(* Logix 5000 project; controller Google vendor 1 type 14 code 151 rev 31.11; software revision 31.00; part 6 of 6 *)
(* tags used below, declared in another part *)
   Alarm : BOOL[64];
   Alarm_Active : BOOL;
   Alarm_Delay : TIMER[32];
   Alarm_Horn : BOOL;
   Alarm_Pulser : Pulser;
   Alarm_Silence : BOOL;
   E_Stop_Pressed : BOOL;
   HMI_Alarm_Silence : BOOL;
   HMI_AutoMode : BOOL;
   HMI_Conv_FWD_Speed : DINT;
   HMI_Conv_REV_Speed : DINT;
   HMI_Conv_Start_Delay : DINT;
   HMI_JogMode : BOOL;
   HMI_ManualMode : BOOL;
   HMI_Output1 : BOOL[32];
   HMI_OutputTest : BOOL[32];
   HMI_PB_Reset : BOOL;
   HMI_System_Full : BOOL;
   Infeed_Conv_Motors : Conveyor_Motor_Control;
   Infeed_ModuleFaultCode : DINT;
   Infeed_Zone1_FWD : BOOL;
   Infeed_Zone1_REV : BOOL;
   Infeed_Zone2_FWD : BOOL;
   Infeed_Zone2_REV : BOOL;
   Infeed_Zone3_FWD : BOOL;
   Infeed_Zone3_REV : BOOL;
   Infeed_Zone4_FWD : BOOL;
   Infeed_Zone4_REV : BOOL;
   L1_Conv_Motors : Conveyor_Motor_Control;
   L1_ModuleFaultCode : DINT;
   L1_Zone1_FWD : BOOL;
   L1_Zone1_REV : BOOL;
   L1_Zone2_FWD : BOOL;
   L1_Zone2_REV : BOOL;
   L1_Zone3_FWD : BOOL;
   L1_Zone3_REV : BOOL;
   L1_Zone4_FWD : BOOL;
   L1_Zone4_REV : BOOL;
   L2_Conv_Motors : Conveyor_Motor_Control;
   L2_ModuleFaultCode : DINT;
   L2_Zone1_FWD : BOOL;
   L2_Zone1_REV : BOOL;
   L2_Zone2_FWD : BOOL;
   L2_Zone2_REV : BOOL;
   L2_Zone3_FWD : BOOL;
   L2_Zone3_REV : BOOL;
   L2_Zone4_FWD : BOOL;
   L2_Zone4_REV : BOOL;
   L3_Conv_Motors : Conveyor_Motor_Control;
   L3_ModuleFaultCode : DINT;
   L3_Zone1_FWD : BOOL;
   L3_Zone1_REV : BOOL;
   L3_Zone2_FWD : BOOL;
   L3_Zone2_REV : BOOL;
   L3_Zone3_FWD : BOOL;
   L3_Zone3_REV : BOOL;
   L3_Zone4_FWD : BOOL;
   L3_Zone4_REV : BOOL;
   L4_Conv_Motors : Conveyor_Motor_Control;
   L4_ModuleFaultCode : DINT;
   L4_Zone1_FWD : BOOL;
   L4_Zone1_REV : BOOL;
   L4_Zone2_FWD : BOOL;
   L4_Zone2_REV : BOOL;
   L4_Zone3_FWD : BOOL;
   L4_Zone3_REV : BOOL;
   L4_Zone4_FWD : BOOL;
   L4_Zone4_REV : BOOL;
   L5_Conv_Motors : Conveyor_Motor_Control;
   L5_ModuleFaultCode : DINT;
   L5_Zone1_FWD : BOOL;
   L5_Zone1_REV : BOOL;
   L5_Zone2_FWD : BOOL;
   L5_Zone2_REV : BOOL;
   L5_Zone3_FWD : BOOL;
   L5_Zone3_REV : BOOL;
   L5_Zone4_FWD : BOOL;
   L5_Zone4_REV : BOOL;
   Level_2_Full : BOOL;
   Level_3_Full : BOOL;
   Level_4_Full : BOOL;
   Level_5_Full : BOOL;
   Lift_Alarm : BOOL;
   Lift_Conv_Motor : Lift_Conv_Motor_Control;
   Lift_ModuleFaultCode : DINT;
   LiftZone_FWD : BOOL;
   LiftZone_REV : BOOL;
   Manual_Mode_Active : BOOL;
   MCR_DelayActive : BOOL;
   MCR_Enable : BOOL;
   MCR_EnableDelay : TIMER;
   MCR_Status : BOOL;
   ONS : DINT[6];
   Outputs_1 : Output_16_Bit;
   PS10017_DC_OK : BOOL;
   Ready_Pulser : Pulser;
   Safety_OK : BOOL;
   Safety_OK_Delay : TIMER;
   Safety_Relay_Status : BOOL;
   Spare_Output : BOOL;
   Stacklight_Amber : BOOL;
   Stacklight_Audible : BOOL;
   Stacklight_Green : BOOL;
   Stacklight_Red : BOOL;
   Starting_Horn : BOOL;
   Starting_Pulser : Pulser;
   Stopping_Pulser : Pulser;
   System : State;
   System_State : DINT;
(* MainProgram, continued *)

ROUTINE R14_Stacklight   (* ladder *)
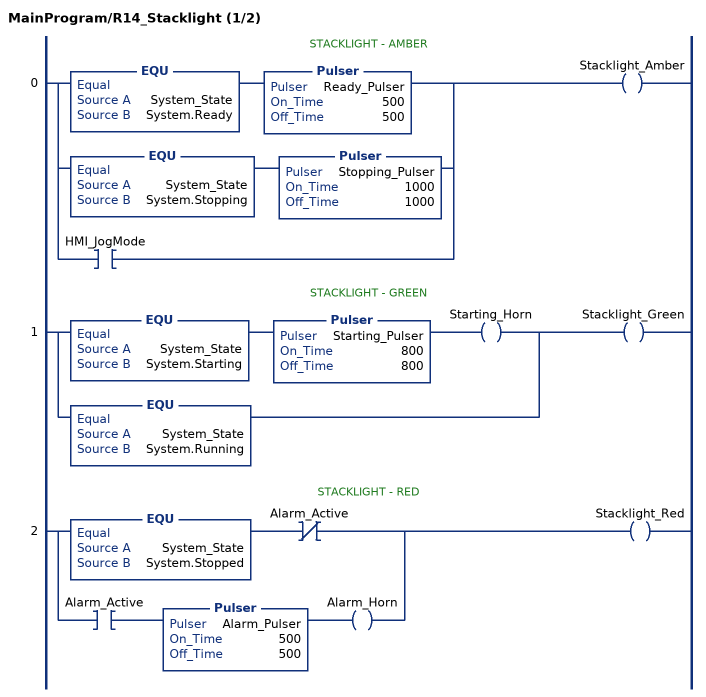
   // STACKLIGHT - AMBER
   0: [EQU(System_State,System.Ready) Pulser(Ready_Pulser,500,500) ,EQU(System_State,System.Stopping) Pulser(Stopping_Pulser,1000,1000) ,XIC(HMI_JogMode) ]OTE(Stacklight_Amber);
   // STACKLIGHT - GREEN
   1: [EQU(System_State,System.Starting) Pulser(Starting_Pulser,800,800) OTE(Starting_Horn) ,EQU(System_State,System.Running) ]OTE(Stacklight_Green);
   // STACKLIGHT - RED
   2: [EQU(System_State,System.Stopped) XIO(Alarm_Active) ,XIC(Alarm_Active) Pulser(Alarm_Pulser,500,500) OTE(Alarm_Horn) ]OTE(Stacklight_Red);
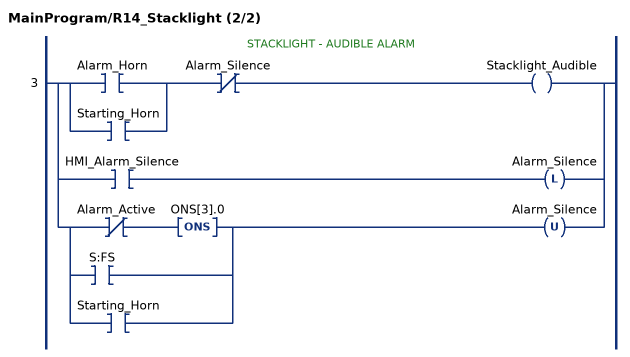
   // STACKLIGHT - AUDIBLE ALARM
   3: [[XIC(Alarm_Horn) ,XIC(Starting_Horn) ] XIO(Alarm_Silence) OTE(Stacklight_Audible) ,XIC(HMI_Alarm_Silence) OTL(Alarm_Silence) ,[XIO(Alarm_Active) ONS(ONS[3].0) ,XIC(S:FS) ,XIC(Starting_Horn) ] OTU(Alarm_Silence) ];
END_ROUTINE

ROUTINE R15_Alarms   (* ladder *)
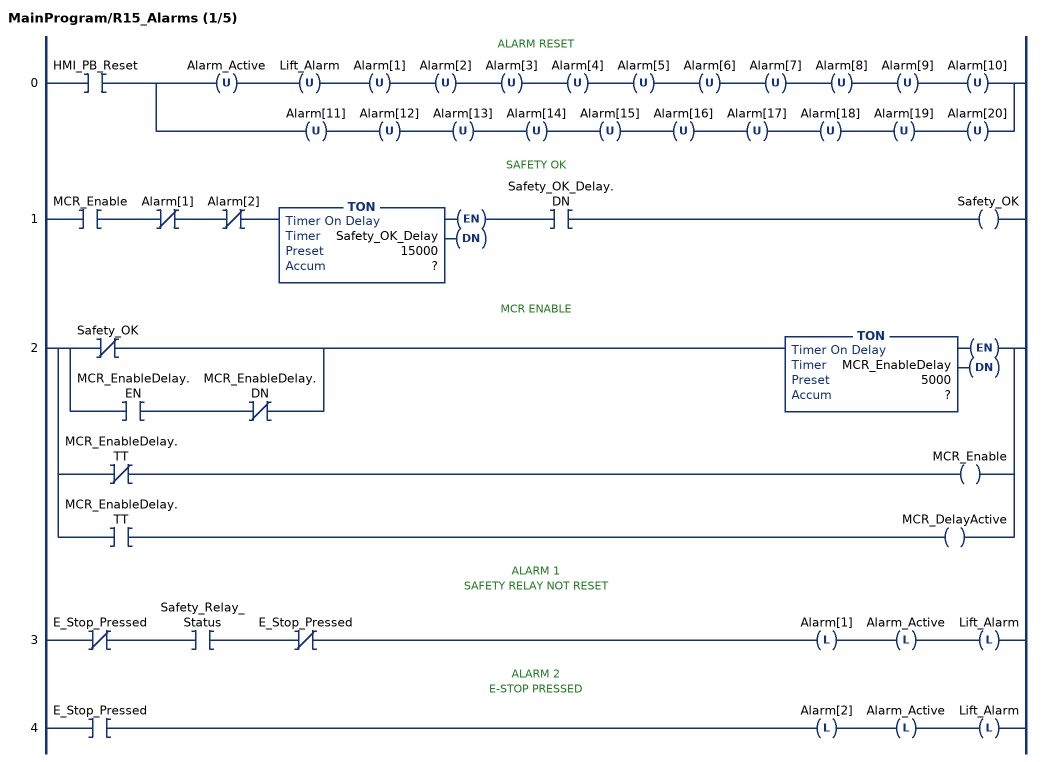
   // ALARM RESET
   0: XIC(HMI_PB_Reset)[OTU(Alarm_Active) OTU(Lift_Alarm) OTU(Alarm[1]) OTU(Alarm[2]) OTU(Alarm[3]) OTU(Alarm[4]) OTU(Alarm[5]) OTU(Alarm[6]) OTU(Alarm[7]) OTU(Alarm[8]) OTU(Alarm[9]) OTU(Alarm[10]) ,OTU(Alarm[11]) OTU(Alarm[12]) OTU(Alarm[13]) OTU(Alarm[14]) OTU(Alarm[15]) OTU(Alarm[16]) OTU(Alarm[17]) OTU(Alarm[18]) OTU(Alarm[19]) OTU(Alarm[20]) ];
   // SAFETY OK
   1: XIC(MCR_Enable)XIO(Alarm[1])XIO(Alarm[2])TON(Safety_OK_Delay,?,?)XIC(Safety_OK_Delay.DN)OTE(Safety_OK);
   // MCR ENABLE
   2: [[XIO(Safety_OK) ,XIC(MCR_EnableDelay.EN) XIO(MCR_EnableDelay.DN) ] TON(MCR_EnableDelay,?,?) ,XIO(MCR_EnableDelay.TT) OTE(MCR_Enable) ,XIC(MCR_EnableDelay.TT) OTE(MCR_DelayActive) ];
   // ALARM 1
   // SAFETY RELAY NOT RESET
   3: XIO(E_Stop_Pressed)XIC(Safety_Relay_Status)XIO(E_Stop_Pressed)OTL(Alarm[1])OTL(Alarm_Active)OTL(Lift_Alarm);
   // ALARM 2
   // E-STOP PRESSED
   4: XIC(E_Stop_Pressed)OTL(Alarm[2])OTL(Alarm_Active)OTL(Lift_Alarm);
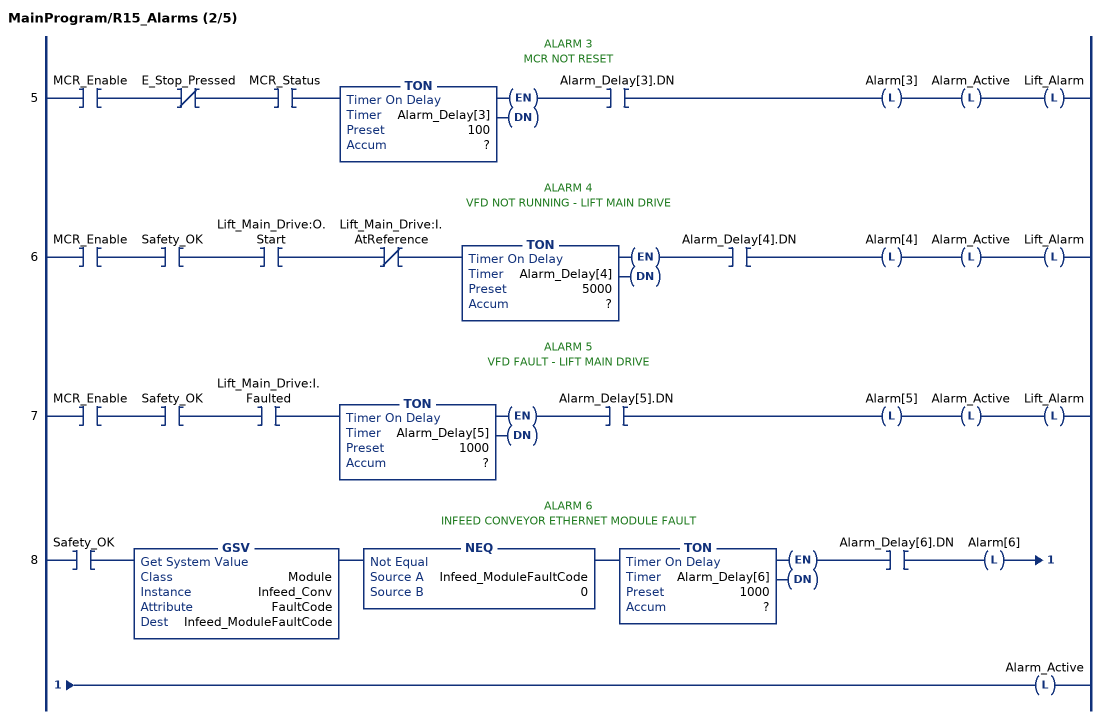
   // ALARM 3
   // MCR NOT RESET
   5: XIC(MCR_Enable)XIO(E_Stop_Pressed)XIC(MCR_Status)TON(Alarm_Delay[3],?,?)XIC(Alarm_Delay[3].DN)OTL(Alarm[3])OTL(Alarm_Active)OTL(Lift_Alarm);
   // ALARM 4
   // VFD NOT RUNNING - LIFT MAIN DRIVE
   6: XIC(MCR_Enable)XIC(Safety_OK)XIC(Lift_Main_Drive:O.Start)XIO(Lift_Main_Drive:I.AtReference)TON(Alarm_Delay[4],?,?)XIC(Alarm_Delay[4].DN)OTL(Alarm[4])OTL(Alarm_Active)OTL(Lift_Alarm);
   // ALARM 5
   // VFD FAULT - LIFT MAIN DRIVE
   7: XIC(MCR_Enable)XIC(Safety_OK)XIC(Lift_Main_Drive:I.Faulted)TON(Alarm_Delay[5],?,?)XIC(Alarm_Delay[5].DN)OTL(Alarm[5])OTL(Alarm_Active)OTL(Lift_Alarm);
   // ALARM 6
   // INFEED CONVEYOR ETHERNET MODULE FAULT
   8: XIC(Safety_OK)GSV(Module,Infeed_Conv,FaultCode,Infeed_ModuleFaultCode)NEQ(Infeed_ModuleFaultCode,0)TON(Alarm_Delay[6],?,?)XIC(Alarm_Delay[6].DN)OTL(Alarm[6])OTL(Alarm_Active);
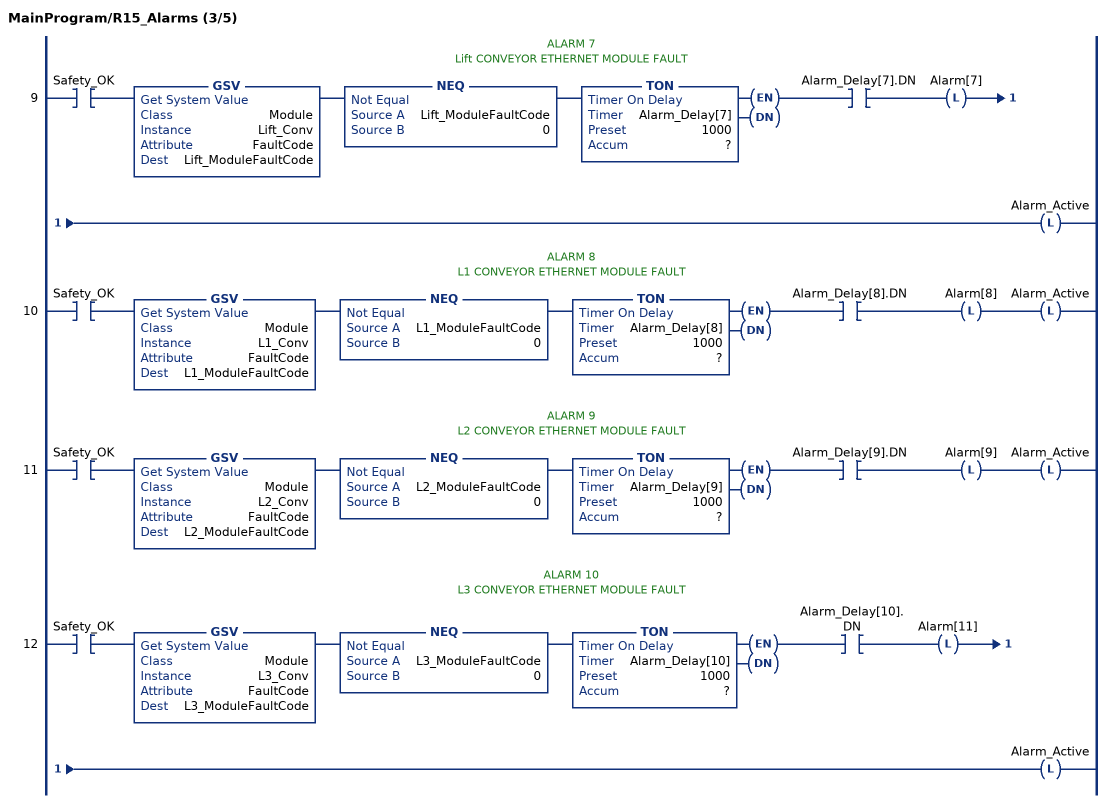
   // ALARM 7
   // Lift CONVEYOR ETHERNET MODULE FAULT
   9: XIC(Safety_OK)GSV(Module,Lift_Conv,FaultCode,Lift_ModuleFaultCode)NEQ(Lift_ModuleFaultCode,0)TON(Alarm_Delay[7],?,?)XIC(Alarm_Delay[7].DN)OTL(Alarm[7])OTL(Alarm_Active);
   // ALARM 8
   // L1 CONVEYOR ETHERNET MODULE FAULT
   10: XIC(Safety_OK)GSV(Module,L1_Conv,FaultCode,L1_ModuleFaultCode)NEQ(L1_ModuleFaultCode,0)TON(Alarm_Delay[8],?,?)XIC(Alarm_Delay[8].DN)OTL(Alarm[8])OTL(Alarm_Active);
   // ALARM 9
   // L2 CONVEYOR ETHERNET MODULE FAULT
   11: XIC(Safety_OK)GSV(Module,L2_Conv,FaultCode,L2_ModuleFaultCode)NEQ(L2_ModuleFaultCode,0)TON(Alarm_Delay[9],?,?)XIC(Alarm_Delay[9].DN)OTL(Alarm[9])OTL(Alarm_Active);
   // ALARM 10
   // L3 CONVEYOR ETHERNET MODULE FAULT
   12: XIC(Safety_OK)GSV(Module,L3_Conv,FaultCode,L3_ModuleFaultCode)NEQ(L3_ModuleFaultCode,0)TON(Alarm_Delay[10],?,?)XIC(Alarm_Delay[10].DN)OTL(Alarm[11])OTL(Alarm_Active);
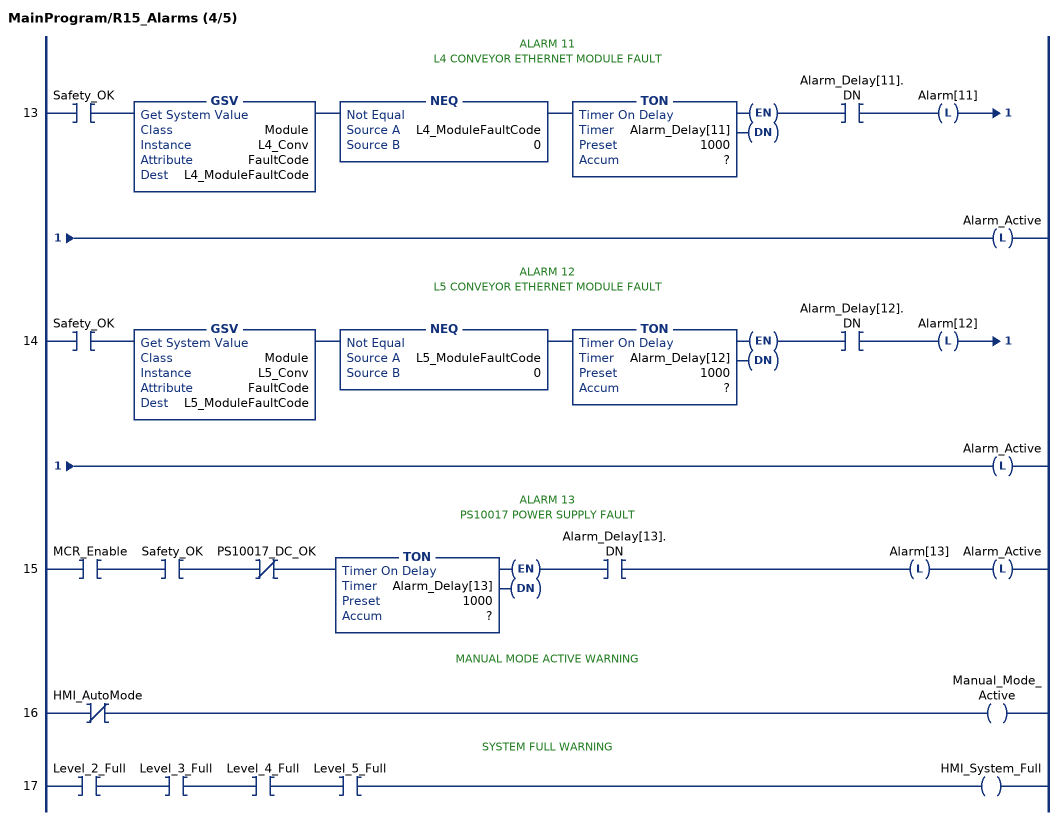
   // ALARM 11
   // L4 CONVEYOR ETHERNET MODULE FAULT
   13: XIC(Safety_OK)GSV(Module,L4_Conv,FaultCode,L4_ModuleFaultCode)NEQ(L4_ModuleFaultCode,0)TON(Alarm_Delay[11],?,?)XIC(Alarm_Delay[11].DN)OTL(Alarm[11])OTL(Alarm_Active);
   // ALARM 12
   // L5 CONVEYOR ETHERNET MODULE FAULT
   14: XIC(Safety_OK)GSV(Module,L5_Conv,FaultCode,L5_ModuleFaultCode)NEQ(L5_ModuleFaultCode,0)TON(Alarm_Delay[12],?,?)XIC(Alarm_Delay[12].DN)OTL(Alarm[12])OTL(Alarm_Active);
   // ALARM 13
   // PS10017 POWER SUPPLY FAULT
   15: XIC(MCR_Enable)XIC(Safety_OK)XIO(PS10017_DC_OK)TON(Alarm_Delay[13],?,?)XIC(Alarm_Delay[13].DN)OTL(Alarm[13])OTL(Alarm_Active);
   // MANUAL MODE ACTIVE WARNING
   16: XIO(HMI_AutoMode)OTE(Manual_Mode_Active);
   // SYSTEM FULL WARNING
   17: XIC(Level_2_Full)XIC(Level_3_Full)XIC(Level_4_Full)XIC(Level_5_Full)OTE(HMI_System_Full);
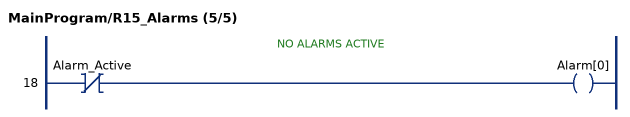
   // NO ALARMS ACTIVE
   18: XIO(Alarm_Active)OTE(Alarm[0]);
END_ROUTINE

ROUTINE R16_Outputs   (* ladder *)
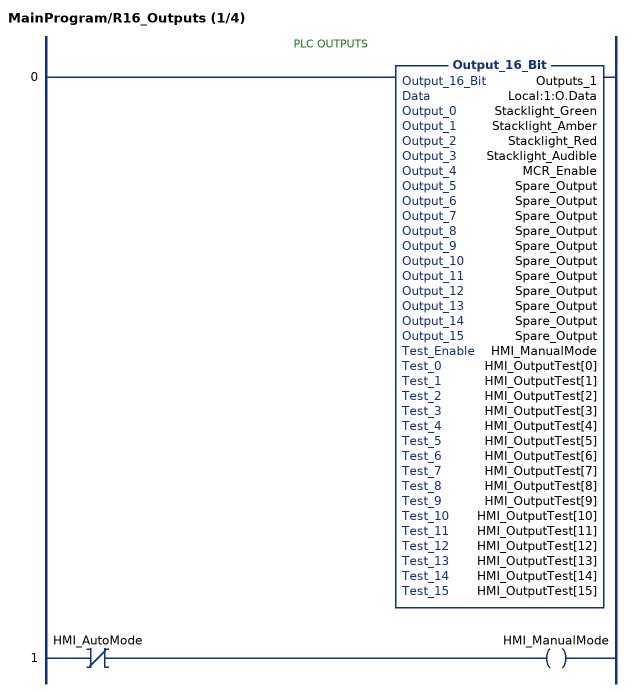
   // PLC OUTPUTS
   0: Output_16_Bit(Outputs_1,Local:1:O.Data,Stacklight_Green,Stacklight_Amber,Stacklight_Red,Stacklight_Audible,MCR_Enable,Spare_Output,Spare_Output,Spare_Output,Spare_Output,Spare_Output,Spare_Output,Spare_Output,Spare_Output,Spare_Output,Spare_Output,Spare_Output,HMI_ManualMode,HMI_OutputTest[0],HMI_OutputTest[1],HMI_OutputTest[2],HMI_OutputTest[3],HMI_OutputTest[4],HMI_OutputTest[5],HMI_OutputTest[6],HMI_OutputTest[7],HMI_OutputTest[8],HMI_OutputTest[9],HMI_OutputTest[10],HMI_OutputTest[11],HMI_OutputTest[12],HMI_OutputTest[13],HMI_OutputTest[14],HMI_OutputTest[15]);
   1: XIO(HMI_AutoMode)OTE(HMI_ManualMode);
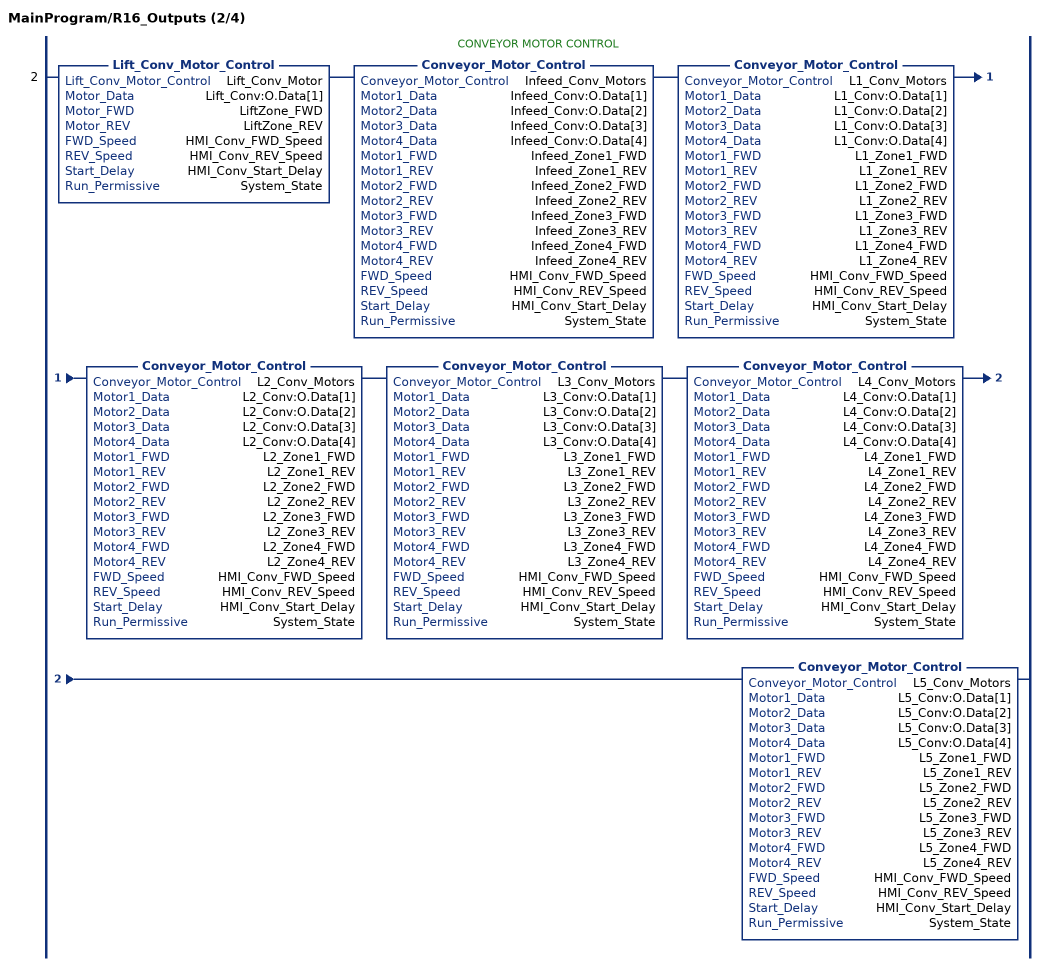
   // CONVEYOR MOTOR CONTROL
   2: Lift_Conv_Motor_Control(Lift_Conv_Motor,Lift_Conv:O.Data[1],LiftZone_FWD,LiftZone_REV,HMI_Conv_FWD_Speed,HMI_Conv_REV_Speed,HMI_Conv_Start_Delay,System_State)Conveyor_Motor_Control(Infeed_Conv_Motors,Infeed_Conv:O.Data[1],Infeed_Conv:O.Data[2],Infeed_Conv:O.Data[3],Infeed_Conv:O.Data[4],Infeed_Zone1_FWD,Infeed_Zone1_REV,Infeed_Zone2_FWD,Infeed_Zone2_REV,Infeed_Zone3_FWD,Infeed_Zone3_REV,Infeed_Zone4_FWD,Infeed_Zone4_REV,HMI_Conv_FWD_Speed,HMI_Conv_REV_Speed,HMI_Conv_Start_Delay,System_State)Conveyor_Motor_Control(L1_Conv_Motors,L1_Conv:O.Data[1],L1_Conv:O.Data[2],L1_Conv:O.Data[3],L1_Conv:O.Data[4],L1_Zone1_FWD,L1_Zone1_REV,L1_Zone2_FWD,L1_Zone2_REV,L1_Zone3_FWD,L1_Zone3_REV,L1_Zone4_FWD,L1_Zone4_REV,HMI_Conv_FWD_Speed,HMI_Conv_REV_Speed,HMI_Conv_Start_Delay,System_State)Conveyor_Motor_Control(L2_Conv_Motors,L2_Conv:O.Data[1],L2_Conv:O.Data[2],L2_Conv:O.Data[3],L2_Conv:O.Data[4],L2_Zone1_FWD,L2_Zone1_REV,L2_Zone2_FWD,L2_Zone2_REV,L2_Zone3_FWD,L2_Zone3_REV,L2_Zone4_FWD,L2_Zone4_REV,HMI_Conv_FWD_Speed,HMI_Conv_REV_Speed,HMI_Conv_Start_Delay,System_State)Conveyor_Motor_Control(L3_Conv_Motors,L3_Conv:O.Data[1],L3_Conv:O.Data[2],L3_Conv:O.Data[3],L3_Conv:O.Data[4],L3_Zone1_FWD,L3_Zone1_REV,L3_Zone2_FWD,L3_Zone2_REV,L3_Zone3_FWD,L3_Zone3_REV,L3_Zone4_FWD,L3_Zone4_REV,HMI_Conv_FWD_Speed,HMI_Conv_REV_Speed,HMI_Conv_Start_Delay,System_State)Conveyor_Motor_Control(L4_Conv_Motors,L4_Conv:O.Data[1],L4_Conv:O.Data[2],L4_Conv:O.Data[3],L4_Conv:O.Data[4],L4_Zone1_FWD,L4_Zone1_REV,L4_Zone2_FWD,L4_Zone2_REV,L4_Zone3_FWD,L4_Zone3_REV,L4_Zone4_FWD,L4_Zone4_REV,HMI_Conv_FWD_Speed,HMI_Conv_REV_Speed,HMI_Conv_Start_Delay,System_State)Conveyor_Motor_Control(L5_Conv_Motors,L5_Conv:O.Data[1],L5_Conv:O.Data[2],L5_Conv:O.Data[3],L5_Conv:O.Data[4],L5_Zone1_FWD,L5_Zone1_REV,L5_Zone2_FWD,L5_Zone2_REV,L5_Zone3_FWD,L5_Zone3_REV,L5_Zone4_FWD,L5_Zone4_REV,HMI_Conv_FWD_Speed,HMI_Conv_REV_Speed,HMI_Conv_Start_Delay,System_State);
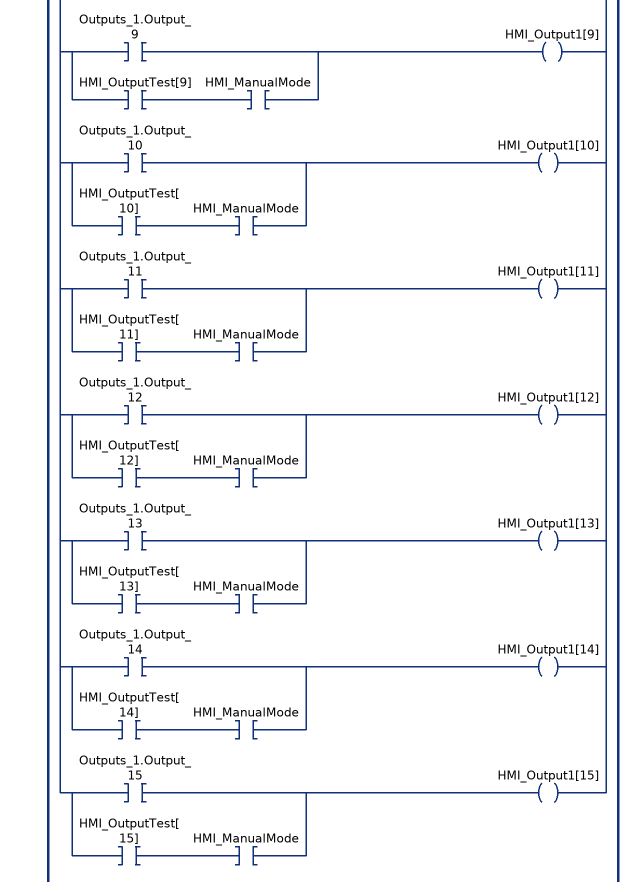
   // HMI OUTPUTS DISPLAY - OUTPUTS 1
   3: [[XIC(Outputs_1.Output_0) ,XIC(HMI_OutputTest[0]) XIC(HMI_ManualMode) ] OTE(HMI_Output1[0]) ,[XIC(Outputs_1.Output_1) ,XIC(HMI_OutputTest[1]) XIC(HMI_ManualMode) ] OTE(HMI_Output1[1]) ,[XIC(Outputs_1.Output_2) ,XIC(HMI_OutputTest[2]) XIC(HMI_ManualMode) ] OTE(HMI_Output1[2]) ,[XIC(Outputs_1.Output_3) ,XIC(HMI_OutputTest[3]) XIC(HMI_ManualMode) ] OTE(HMI_Output1[3]) ,[XIC(Outputs_1.Output_4) ,XIC(HMI_OutputTest[4]) XIC(HMI_ManualMode) ] OTE(HMI_Output1[4]) ,[XIC(Outputs_1.Output_5) ,XIC(HMI_OutputTest[5]) XIC(HMI_ManualMode) ] OTE(HMI_Output1[5]) ,[XIC(Outputs_1.Output_6) ,XIC(HMI_OutputTest[6]) XIC(HMI_ManualMode) ] OTE(HMI_Output1[6]) ,[XIC(Outputs_1.Output_7) ,XIC(HMI_OutputTest[7]) XIC(HMI_ManualMode) ] OTE(HMI_Output1[7]) ,[XIC(Outputs_1.Output_8) ,XIC(HMI_OutputTest[8]) XIC(HMI_ManualMode) ] OTE(HMI_Output1[8]) ,[XIC(Outputs_1.Output_9) ,XIC(HMI_OutputTest[9]) XIC(HMI_ManualMode) ] OTE(HMI_Output1[9]) ,[XIC(Outputs_1.Output_10) ,XIC(HMI_OutputTest[10]) XIC(HMI_ManualMode) ] OTE(HMI_Output1[10]) ,[XIC(Outputs_1.Output_11) ,XIC(HMI_OutputTest[11]) XIC(HMI_ManualMode) ] OTE(HMI_Output1[11]) ,[XIC(Outputs_1.Output_12) ,XIC(HMI_OutputTest[12]) XIC(HMI_ManualMode) ] OTE(HMI_Output1[12]) ,[XIC(Outputs_1.Output_13) ,XIC(HMI_OutputTest[13]) XIC(HMI_ManualMode) ] OTE(HMI_Output1[13]) ,[XIC(Outputs_1.Output_14) ,XIC(HMI_OutputTest[14]) XIC(HMI_ManualMode) ] OTE(HMI_Output1[14]) ,[XIC(Outputs_1.Output_15) ,XIC(HMI_OutputTest[15]) XIC(HMI_ManualMode) ] OTE(HMI_Output1[15]) ];
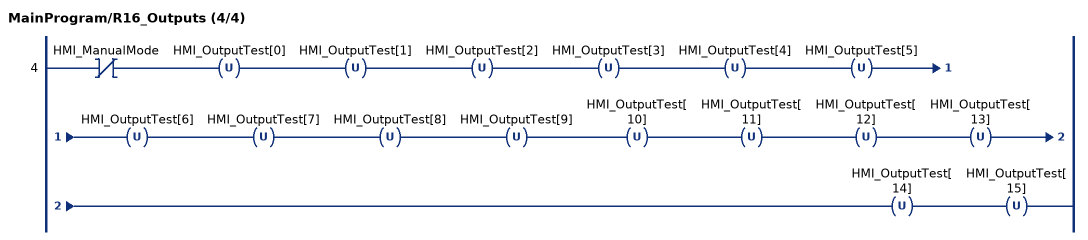
   4: XIO(HMI_ManualMode)OTU(HMI_OutputTest[0])OTU(HMI_OutputTest[1])OTU(HMI_OutputTest[2])OTU(HMI_OutputTest[3])OTU(HMI_OutputTest[4])OTU(HMI_OutputTest[5])OTU(HMI_OutputTest[6])OTU(HMI_OutputTest[7])OTU(HMI_OutputTest[8])OTU(HMI_OutputTest[9])OTU(HMI_OutputTest[10])OTU(HMI_OutputTest[11])OTU(HMI_OutputTest[12])OTU(HMI_OutputTest[13])OTU(HMI_OutputTest[14])OTU(HMI_OutputTest[15]);
END_ROUTINE
END_PROGRAM
